{attribute addProperty BoxType "EPP1321-0060-0016"}
{attribute addProperty Id "InfoDataInfoData_192954DE162"}
{attribute addProperty CRC "395970889"}
{attribute addProperty SizeInBites "16"}
{attribute addProperty SizeInBytes "2"}
TYPE EPP1321_179A0949 :
STRUCT
	{attribute addProperty Name "InfoData"}
	InfoData : InfoData_192954DE;
END_STRUCT
END_TYPE

(* stored: Version 1.2.0.0, ProductVersion 3.1.4024.9
   DUT EPP1321_179A0949: Id {a15740bb-9fbb-4b9c-b2cb-7f743f62555b} *)
